// SIMATIC S7-200 project (STEP 7-Micro/WIN), CPU 221 REL 01.10

ORGANIZATION_BLOCK 主程序:OB1
TITLE=程序注释
BEGIN
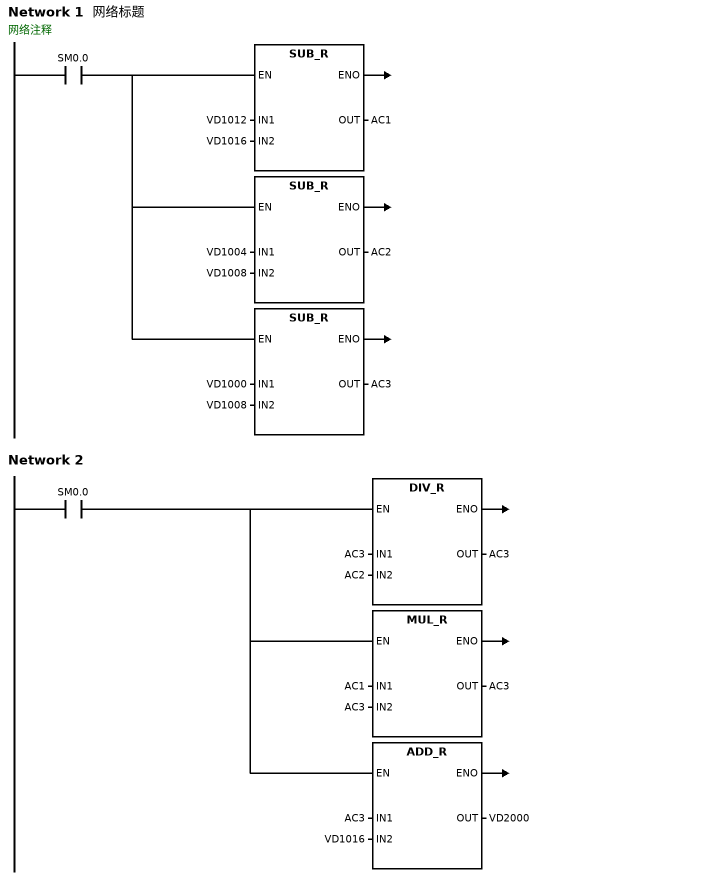
Network 1 // 网络标题
// 网络注释
LD     SM0.0
MOVR   VD1012, AC1
-R     VD1016, AC1
MOVR   VD1004, AC2
-R     VD1008, AC2
MOVR   VD1000, AC3
-R     VD1008, AC3
Network 2
// (network saved uncompiled; LAD cells follow)
// row 0: c0 -| |- SM0.0  c1 -- v  c2 --  c3 [DIV_R EN:=power@row0, IN1:=AC3, IN2:=AC2, ENO=>power, OUT=>AC3]  c4 ->
// row 1: c1 ^v  c3 [box]
// row 2: c1 ^v  c2 --  c3 [MUL_R EN:=power@row2, IN1:=AC1, IN2:=AC3, ENO=>power, OUT=>AC3]  c4 ->
// row 3: c1 ^v  c3 [box]
// row 4: c1 ^  c2 --  c3 [ADD_R EN:=power@row4, IN1:=AC3, IN2:=VD1016, ENO=>power, OUT=>VD2000]  c4 ->
// row 5: c3 [box]
END_ORGANIZATION_BLOCK
